// TIA Portal project "garajoto" (V20)

(* hardware
DEVICE "S7-1200 station_1"  S7-1200 Station
   slot 0: "Rack_0"  S7-1200 Rack  Rack  V1.0
   slot 1: "PLC_1"  CPU 1212C DC/DC/DC  6ES7 212-1AE40-0XB0  V4.7
*)

// ===== PLC "PLC_1"  CPU 1212C DC/DC/DC =====

VAR_GLOBAL   // PLC tag table "Default tag table"
   "man-oto" AT %I0.0 : Bool;
   "man aç" AT %I0.1 : Bool;
   "man kapa" AT %I0.2 : Bool;
   "fotosel1" AT %I0.3 : Bool;
   "fotosel2" AT %I0.4 : Bool;
   "kapı aç switch" AT %I0.5 : Bool;
   "kapı kapalı switch" AT %I0.6 : Bool;
   "kapı açma valve" AT %Q0.0 : Bool;
   "kapı kapatma valve" AT %Q0.1 : Bool;
   "oto çalışma mem" AT %M10.0 : Bool;
   "man aç mem" AT %M10.1 : Bool;
   "man kapa mem" AT %M10.2 : Bool;
   "oto aç mem" AT %M10.3 : Bool;
   "oto kapat mem" AT %M10.4 : Bool;
END_VAR

// folder: System blocks/Program resources

DATA_BLOCK "timer1"   // DB1
{ S7_Optimized_Access := 'TRUE' }
AUTHOR : Simatic
FAMILY : IEC
NAME : IEC_TMR
VERSION : 1.0
// stored: InstanceOfName IEC_TIMER
"IEC_TIMER"
BEGIN
END_DATA_BLOCK

// folder: (top level)

ORGANIZATION_BLOCK "Main"   // OB1, LAD, ProgramCycle
TITLE = "Main Program Sweep (Cycle)"
{ S7_Optimized_Access := 'TRUE' }
VERSION : 0.1
   VAR_INPUT
      Initial_Call : Bool;   // Initial call of this OB
      Remanence : Bool;   // =True, if remanent data are available
   END_VAR
BEGIN

REGION Network 1
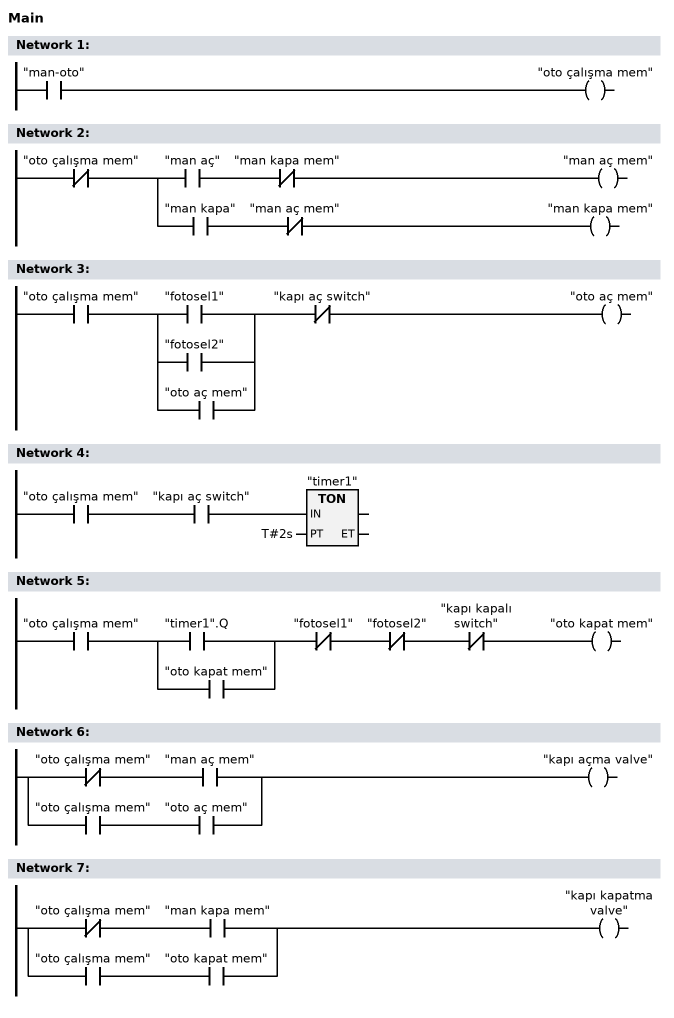
   RUNG wire#powerrail
      Contact( "man-oto" )
      Coil( "oto çalışma mem" )
   END_RUNG
   // the same network as SCL:
   "oto çalışma mem" := "man-oto";
END_REGION

REGION Network 2
   RUNG wire#powerrail
      I_Contact( "oto çalışma mem" )
      wire#w1
      Contact( "man aç" )
      I_Contact( "man kapa mem" )
      Coil( "man aç mem" )
   END_RUNG
   RUNG wire#w1
      Contact( "man kapa" )
      I_Contact( "man aç mem" )
      Coil( "man kapa mem" )
   END_RUNG
   // the same network as SCL:
   "man aç mem" := NOT "oto çalışma mem" AND "man aç" AND NOT "man kapa mem";
   "man kapa mem" := NOT "oto çalışma mem" AND "man kapa" AND NOT "man aç mem";
END_REGION

REGION Network 3
   RUNG wire#powerrail
      Contact( "oto çalışma mem" )
      wire#w1
      Contact( "fotosel1" )
      wire#w2
      I_Contact( "kapı aç switch" )
      Coil( "oto aç mem" )
   END_RUNG
   RUNG wire#w1
      Contact( "fotosel2" )
   END_RUNG wire#w2
   RUNG wire#w1
      Contact( "oto aç mem" )
   END_RUNG wire#w2
   // the same network as SCL:
   "oto aç mem" := "oto çalışma mem" AND ("fotosel1" OR "fotosel2" OR "oto aç mem") AND NOT "kapı aç switch";
END_REGION

REGION Network 4
   "timer1".TON(IN := "oto çalışma mem" AND "kapı aç switch", PT := T#2s);
END_REGION

REGION Network 5
   RUNG wire#powerrail
      Contact( "oto çalışma mem" )
      wire#w1
      Contact( "timer1".Q )
      wire#w2
      I_Contact( "fotosel1" )
      I_Contact( "fotosel2" )
      I_Contact( "kapı kapalı switch" )
      Coil( "oto kapat mem" )
   END_RUNG
   RUNG wire#w1
      Contact( "oto kapat mem" )
   END_RUNG wire#w2
   // the same network as SCL:
   "oto kapat mem" := "oto çalışma mem" AND ("timer1".Q OR "oto kapat mem") AND NOT "fotosel1" AND NOT "fotosel2" AND NOT "kapı kapalı switch";
END_REGION

REGION Network 6
   RUNG wire#powerrail
      I_Contact( "oto çalışma mem" )
      Contact( "man aç mem" )
      wire#w1
      Coil( "kapı açma valve" )
   END_RUNG
   RUNG wire#powerrail
      Contact( "oto çalışma mem" )
      Contact( "oto aç mem" )
   END_RUNG wire#w1
   // the same network as SCL:
   "kapı açma valve" := (NOT "oto çalışma mem" AND "man aç mem") OR ("oto çalışma mem" AND "oto aç mem");
END_REGION

REGION Network 7
   RUNG wire#powerrail
      I_Contact( "oto çalışma mem" )
      Contact( "man kapa mem" )
      wire#w1
      Coil( "kapı kapatma valve" )
   END_RUNG
   RUNG wire#powerrail
      Contact( "oto çalışma mem" )
      Contact( "oto kapat mem" )
   END_RUNG wire#w1
   // the same network as SCL:
   "kapı kapatma valve" := (NOT "oto çalışma mem" AND "man kapa mem") OR ("oto çalışma mem" AND "oto kapat mem");
END_REGION
END_ORGANIZATION_BLOCK